// TwinCAT 3 PLC project GEMMA
// ProgramVersion: 3.1.4023.0
// libraries:
//   Tc2_Standard, * (Beckhoff Automation GmbH)
//   Tc2_System, * (Beckhoff Automation GmbH)
//   Tc3_Module, * (Beckhoff Automation GmbH)
//   VisuDialogs, * (System)
// project tree:
//   DUTs/ E_GEMMA.TcTLEO
//   / GlobalTextList.TcGTLO, ModoDescripcion.TcTLO, PlcTask.TcTTO, Visualization Manager.TcVMO (not stored)
//   POUs/Estacion/ FB_Estacion.TcPOU, FB_Coordinador_SFC.TcPOU, FB_Director.TcPOU
//   POUs/FBs/ FB_Clock.TcPOU
//   POUs/ MAIN.TcPOU
//   POUs/Tareas/ FB_CintaSituarPale_SFC.TcPOU, FB_CintaTransferirPale_SFC.TcPOU, FB_EstacionFinalizar_SFC.TcPOU, FB_EstacionPreparar_SFC.TcPOU, FB_EstacionRestaurar_SFC.TcPOU, FB_ManipuladorCargarBase_SFC.TcPOU, FB_ManipuladorDescargarBase_SFC.TcPOU, FB_PrensaPrensarRodamiento_SFC.TcPOU
//   VISUs/ TC_VISU.TcVIS

CONFIGURATION GEMMA
    RESOURCE PLC ON TwinCAT3
        TASK PlcTask(INTERVAL := T#10ms, PRIORITY := 24);
        PROGRAM MAIN WITH PlcTask : MAIN;
    END_RESOURCE
END_CONFIGURATION

// ---- DUTs/E_GEMMA.TcTLEO
{attribute 'qualified_only'}
{attribute 'strict'}
TYPE E_GEMMA :
(
    // Modos de la Guia de Estudio de los Modos de Marcha y Parada
    // [Modes du Guide d'Etude des Modes de Marche et d'Arrêt]
    // [Modes of Study Guide of the Modes of Operating and Stopping]

    // Procedimientos de parada [Les procédures d'arrets - Stop procedures]
    A1, //  0: Parada en el estado inicial [Arrêt dans etat initial - Stopped in the initial state]
    A2, //  1: Parada solicitada a final de ciclo [Arret demandé en fin de cycle - Requested end cycle stop]
    A3, //  2: Parada solicitada en un estado determinado [Arret demande dans etat determine - Requested particular state stop]
    A4, //  3: Parada obtenida [Arret obtenu - Obteined stop]
    A5, //  4: Preparacion para la recuperacion del fallo [Preparation pour remise en route apres defaillance - Preparation for the recovery of the failure]
    A6, //  5: Situando la PO en el estado inicial [Mise PO dans état initial - Set the PO in initial state]
    A7, //  6: Situando la PO en un estado determinado [Mise PO dans état déterminé - Set the PO in a certain state]

    // Procedimientos de funcionamiento [Les procédures de fonctionnement - Operating procedures]
    F1, //  7: Produccion normal [Production normale - Normal operation]
    F2, //  8: Secuencia de preparacion [Marche de preparation - Preparation sequence]
    F3, //  9: Secuencia de finalizacion [Marche de cloture - Ending sequence]
    F4, // 10: Verificacion en desorden [Marche de verification dans le desordre - Verification with no order]
    F5, // 11: Verificacion en orden [Marche de verification dans l'ordre - Verification whit order]
    F6, // 12: Secuencia de prueba [Marche de test - Test sequence]

    // Procedimientos de fallo [Les procédures en défaillances - Failure procedures]
    D1, // 13: Parada de emergencia [Arret d'urgence - Emergency stop]
    D2, // 14: Diagnostico y/o tratamiento de los fallos [Diagnostic et/ou traitement de la défaillance - Diagnosis and/or treatment of failures]
    D3  // 15: Produccion a pesar de los fallos [Production tout de même - Production despite the failures]
);
END_TYPE

// ---- POUs/MAIN.TcPOU
PROGRAM MAIN
VAR
    Estacion: FB_Estacion;
END_VAR

Estacion();

END_PROGRAM

// ---- POUs/Estacion/FB_Estacion.TcPOU
FUNCTION_BLOCK FB_Estacion
VAR_INPUT
    EstadoPausa: BOOL;
    EstadoReinicia: BOOL;
    UnidadesSolicitadas: UINT := 1;
    
    RodamientoBajo: BOOL;
    TpoCintaRetenedor: TIME := T#1S;
    TpoCintaSeparador: TIME := T#1S;
    TpoPaleEntrada: TIME := T#400ms;
    TpoPaleSalida: TIME := T#1s;
    TpoPaleTransferencia: TIME := T#1S;
    TpoPrensaHidraulico: TIME := T#2s;
    TpoPrensaProtector: TIME := T#2s;
END_VAR
VAR_OUTPUT
    CondicionInicial: BOOL := TRUE;
    UnidadesPendientes: UINT;
    UnidadesRealizadas: UINT;
    PaleCodigo: BYTE;
    
    // Entradas comunes
    PulsadorEmergencia AT %I*: BOOL;
    SelectorManual AT %I*: BOOL;
    PulsadorMarcha AT %I*: BOOL;
    PulsadorParada AT %I*: BOOL := TRUE; // Contacto normalmente cerrado
    EstacionConectada AT %I*: BOOL := TRUE;
    DetectorPresion AT %I*: BOOL := TRUE;

    PalePresencia AT %I*: BOOL;
    PaleCodigoBit0 AT %I*: BOOL;
    PaleCodigoBit1 AT %I*: BOOL;
    PaleCodigoBit2 AT %I*: BOOL;

    // Entradas espeficicas
    ManipuladorDetras AT %I*: BOOL; // Sobre el pale
    ManipuladorMedio AT %I*: BOOL := TRUE; // En la vertical
    ManipuladorDelante AT %I*: BOOL; // Sobre el punto de trasvase de la presa
    IntroductorDetras AT %I*: BOOL := TRUE;
    IntroductorDelante AT %I*: BOOL;
    ExtractorDetras AT %I*: BOOL := TRUE;
    ExtractorDelante AT %I*: BOOL;
    ProtectorAbajo AT %I*: BOOL;
    PrensadorArriba AT %I*: BOOL := TRUE;
    PrensadorAbajoAlto AT %I*: BOOL;
    PrensadorAbajoBajo AT %I*: BOOL;
    ManipuladorVacioObtenido AT %I*: BOOL;
END_VAR
VAR
    ModoAnterior: E_GEMMA;
    
    // Bloques funcionales
    CLK: FB_Clock;
    Director: FB_Director;
    Coordinador: FB_Coordinador_SFC;
    Restaurar: FB_EstacionRestaurar_SFC;
    Preparar: FB_EstacionPreparar_SFC;
    Finalizar: FB_EstacionFinalizar_SFC;
    SituarPale: FB_CintaSituarPale_SFC;
    CargarBase: FB_ManipuladorCargarBase_SFC;
    PrensarRodamiento: FB_PrensaPrensarRodamiento_SFC;
    DescargarBase: FB_ManipuladorDescargarBase_SFC;
    TransferirPale: FB_CintaTransferirPale_SFC;
    
    // Salidas comunes
    DesconectaEstacion AT %Q*: BOOL;
    LamparaAlarma AT %Q*: BOOL;
    LamparaMarcha AT %Q*: BOOL;
    AvisadorSonoro AT %Q*: BOOL;

    CintaMotorActiva AT %Q*: BOOL;
    CintaMotorInvierte AT %Q*: BOOL;
    CintaRetenedorBaja AT %Q*: BOOL;
    CintaSeparadorSube AT %Q*: BOOL;
    
    // Salidas especificas
    ManipuladorAdelante AT %Q*: BOOL; // Hacia el punto de trasvase de la prensa
    ManipuladorAtras AT %Q*: BOOL; // Hacia el pale
    IntroductorAdelante AT %Q*: BOOL;
    ExtractorAdelante AT %Q*: BOOL;
    ProtectorBaja AT %Q*: BOOL;
    PrensadorBaja AT %Q*: BOOL;
    PrensadorSube AT %Q*: BOOL;
    ManipuladorSucciona AT %Q*: BOOL;
    HidraulicoActiva AT %Q*: BOOL;
END_VAR

// MODO AUTOMATICO
CLK();

Director(
    CondicionInicial := CondicionInicial,
    CondicionMarcha := (UnidadesSolicitadas > 0) AND CondicionInicial,
    Emergencia := PulsadorEmergencia,
    Finalizada := Finalizar.Done,
    FinTarea := (UnidadesPendientes = 0),
    FinCiclo := Coordinador.Done,
    Manual := SelectorManual,
    Marcha := PulsadorMarcha,
    ParaCiclo := NOT PulsadorParada,
    Preparada := Preparar.Done,
    Reinicia := EstadoReinicia
    );

IF (Director.Modo <> E_GEMMA.F4) THEN
    // Bloques funcionales     
    Restaurar(
        SFCPause := NOT EstadoReinicia AND EstadoPausa,
        SFCReset := EstadoReinicia,
        Ack := TRUE ,
        Execute := (Director.Modo = E_GEMMA.A6) AND PulsadorMarcha,
        ManipuladorDetras := ManipuladorDetras,
        ManipuladorMedio := ManipuladorMedio,
        PrensadorArriba := PrensadorArriba
        );
        
    Preparar(
        SFCPause := NOT EstadoReinicia AND EstadoPausa,
        SFCReset := EstadoReinicia,
        Ack := (Director.Modo <> E_GEMMA.F2),
        Execute := (Director.Modo = E_GEMMA.F2),
        );

    Finalizar(
        SFCPause := NOT EstadoReinicia AND EstadoPausa,
        SFCReset := EstadoReinicia,
        Ack := (Director.Modo <> E_GEMMA.F3),
        Execute := (Director.Modo = E_GEMMA.F3),
        );
    
    Coordinador(
        UnidadesPendientes := UnidadesPendientes,
        UnidadesRealizadas := UnidadesRealizadas,
        SFCPause := NOT EstadoReinicia AND EstadoPausa,
        SFCReset := EstadoReinicia,
        Ack := TRUE,
        Execute := (Director.Modo = E_GEMMA.F1),
        PaleSituado := SituarPale.Done,
        BaseCargada := CargarBase.Done,
        RodamientoPrensado := PrensarRodamiento.Done,
        BaseDescargada := DescargarBase.Done,
        PaleTransferido := TransferirPale.Done
        );
        
    SituarPale(
        SFCPause := NOT EstadoReinicia AND EstadoPausa,
        SFCReset := EstadoReinicia,
        Ack := NOT Coordinador.SituaPale,
        Execute := Coordinador.SituaPale,
        TpoPaleEntrada := TpoPaleEntrada,
        PalePresencia := PalePresencia,
        PaleCodigoBit0 := PaleCodigoBit0,
        PaleCodigoBit1 := PaleCodigoBit1,
        PaleCodigoBit2:= PaleCodigoBit2
        );
        
    CargarBase(
        SFCPause := NOT EstadoReinicia AND EstadoPausa,
        SFCReset := EstadoReinicia,
        Ack := NOT Coordinador.CargaBase,
        Execute := Coordinador.CargaBase,
        ManipuladorDetras := ManipuladorDetras,
        ManipuladorMedio := ManipuladorMedio,
        ManipuladorDelante := ManipuladorDelante,
        ManipuladorVacioObtenido := ManipuladorVacioObtenido
        );
    
    PrensarRodamiento(
        SFCPause := NOT EstadoReinicia AND EstadoPausa,
        SFCReset := EstadoReinicia,
        Ack := NOT Coordinador.PrensaRodamiento,
        Execute := Coordinador.PrensaRodamiento,
        RodamientoBajo := RodamientoBajo,
        TpoPrensaHidraulico := TpoPrensaHidraulico,
        TpoPrensaProtector := TpoPrensaProtector,
        IntroductorDetras := IntroductorDetras,
        IntroductorDelante := IntroductorDelante,
        ExtractorDetras := ExtractorDetras,
        ExtractorDelante := ExtractorDelante,
        ProtectorAbajo := ProtectorAbajo,
        PrensadorArriba := PrensadorArriba,
        PrensadorAbajoAlto := PrensadorAbajoAlto,
        PrensadorAbajoBajo := PrensadorAbajoBajo
        );
    
    DescargarBase(
        SFCPause := NOT EstadoReinicia AND EstadoPausa,
        SFCReset := EstadoReinicia,
        Ack := NOT Coordinador.DescargaBase,
        Execute := Coordinador.DescargaBase,
        ManipuladorDetras := ManipuladorDetras,
        ManipuladorMedio := ManipuladorMedio,
        ManipuladorDelante := ManipuladorDelante,
        ManipuladorVacioObtenido := ManipuladorVacioObtenido
        );
    
    TransferirPale(
        SFCPause := NOT EstadoReinicia AND EstadoPausa,
        SFCReset := EstadoReinicia,
        Ack := NOT Coordinador.TransfierePale,
        Execute := Coordinador.TransfierePale,
        TpoCintaRetenedor := TpoCintaRetenedor,
        TpoCintaSeparador := TpoCintaSeparador,
        TpoPaleSalida := TpoPaleSalida,
        TpoPaleTransferencia := TpoPaleTransferencia,
        PalePresencia := PalePresencia
        );
    
    // Acciones
    // DesconectaEstacion :=
    LamparaAlarma := (Director.Modo = E_GEMMA.D1) OR ((Director.Modo = E_GEMMA.A6) AND CLK.Q);
    LamparaMarcha := Director.Produccion OR ((Director.Modo = E_GEMMA.A1) AND CLK.Q);
    AvisadorSonoro := ((Director.Modo = E_GEMMA.F2) AND CLK.Q) OR (Director.Modo = E_GEMMA.F3); 

    CintaMotorActiva := NOT EstadoPausa AND (SituarPale.CintaMotorActiva OR TransferirPale.CintaMotorActiva);
    // CintaMotorInvierte :=
    CintaRetenedorBaja:= TransferirPale.CintaRetenedorBaja;
    CintaSeparadorSube :=TransferirPale.CintaSeparadorSube;
    ManipuladorAdelante := CargarBase.ManipuladorAdelante OR DescargarBase.ManipuladorAdelante OR Restaurar.ManipuladorAdelante;
    ManipuladorAtras := CargarBase.ManipuladorAtras OR DescargarBase.ManipuladorAtras OR Restaurar.ManipuladorAtras;
    IntroductorAdelante := PrensarRodamiento.IntroductorAdelante;
    ExtractorAdelante := PrensarRodamiento.ExtractorAdelante;
    ProtectorBaja := PrensarRodamiento.ProtectorBaja;
    PrensadorBaja := PrensarRodamiento.PrensadorBaja;
    PrensadorSube := PrensarRodamiento.PrensadorSube OR Restaurar.PrensadorSube;
    ManipuladorSucciona := CargarBase.ManipuladorSucciona OR DescargarBase.ManipuladorSucciona;
    HidraulicoActiva := PrensarRodamiento.HidraulicoActiva;
END_IF

// Parametros de Salida
CondicionInicial := EstacionConectada AND ManipuladorMedio AND IntroductorDetras AND ExtractorDetras AND PrensadorArriba;

// Al iniciar una tarea (abandonar modo A1) se actualiza las unidades pendientes
IF ((ModoAnterior = E_GEMMA.A1) AND (Director.Modo <> E_GEMMA.A1) AND (UnidadesPendientes = 0)) THEN
    UnidadesPendientes := UnidadesSolicitadas;
END_IF
 
IF (Director.Modo <> E_GEMMA.F4) THEN
    PaleCodigo := SituarPale.PaleCodigo;
ELSE 
    PaleCodigo.0 := PaleCodigoBit0;
    PaleCodigo.1 := PaleCodigoBit1;
    PaleCodigo.2 := PaleCodigoBit2;
END_IF

// ACTULIZACION DE IMAGENES
ModoAnterior := Director.Modo;

END_FUNCTION_BLOCK

// ---- POUs/FBs/FB_Clock.TcPOU
FUNCTION_BLOCK FB_Clock
(*
Square wave oscillator

Copyright (c) 2009-2017 victortorreslopez

GNU General Public License

Version history
2.1, 2017/03/15, VTL: style review (PLCopen Coding Guidelines)
2.0, 2014/12/29, VTL: complete review
1.0, 2009/11/06, VTL: first release
0.0, 2009/11/06, VTL: alfa release
*)
VAR_INPUT
  EN: BOOL := TRUE;	(* ENabled *)
  PT: TIME := T#500ms; (* Semicycle time *)
END_VAR
VAR_OUTPUT
  ET: TIME; (* Elapsed time *)
  Q: BOOL; (* Square wave *)
END_VAR
VAR
  Timer: TON; (* Auto-pilot timer *)
END_VAR

(* OUTPUT FUNCTION *)
IF Timer.Q THEN
  Q := NOT Q;
END_IF

(* FUNCTION BLOCKS *)
Timer(IN := EN AND NOT Timer.Q, PT := PT, ET => ET);

END_FUNCTION_BLOCK

// ---- POUs/Estacion/FB_Director.TcPOU
FUNCTION_BLOCK FB_Director
VAR_INPUT
    CondicionInicial: BOOL; // Condiciones materiales necesarias para iniciar la produccion
    CondicionMarcha: BOOL; // Condiciones logicas necesarias para iniciar la produccion
    Emergencia: BOOL;
    Finalizada: BOOL;
    FinTarea: BOOL;
    FinCiclo: BOOL;
    Manual: BOOL;
    Marcha: BOOL;
    ParaCiclo: BOOL;
    Preparada: BOOL;
    Reinicia: BOOL;
END_VAR
VAR_OUTPUT
    Modo: E_GEMMA := E_GEMMA.A6;

    Defecto: BOOL; // Procedimientos de defecto
    Funcionamiento: BOOL; // Procedimientos de funcionamiento
    Parada: BOOL; // Procedimientos de parada
    Produccion: BOOL; // Procedimientos que proporcionan valor añadido
END_VAR

// FUNCION DE ESTADO
IF Emergencia THEN
    Modo := E_GEMMA.D1;
ELSIF Reinicia THEN
    Modo := E_GEMMA.A6;
ELSE
    CASE Modo OF
        // Procedimientos de parada
        E_GEMMA.A1: // Parada en el estado inicial
            IF NOT CondicionInicial THEN
                Modo := E_GEMMA.A6;
            ELSIF Manual THEN
                Modo := E_GEMMA.F4;
            ELSIF (CondicionMarcha AND Marcha) THEN
                Modo := E_GEMMA.F2;
            END_IF
        E_GEMMA.A2: // Parada solicitada a final de ciclo
            IF FinCiclo THEN
                Modo := E_GEMMA.A1;
            END_IF
        E_GEMMA.A3: // Parada solicitada en un estado determinado 
            ;
        E_GEMMA.A4: // Parada obtenida 
            ;
        E_GEMMA.A5: // Preparando de reanudacion tras el fallo 
            ;
        E_GEMMA.A6: // Situando la PO en el estado inicial 
            IF CondicionInicial THEN
                Modo := E_GEMMA.A1;
            ELSIF Manual THEN
                Modo := E_GEMMA.F4;
            END_IF
        E_GEMMA.A7: // Situando la PO en un estado determinado 
            ;

        // Procedimientos de funcionamiento 
        E_GEMMA.F1: // Produccion normal 
            IF FinTarea THEN
                Modo := E_GEMMA.F3;
            ELSIF ParaCiclo THEN
                Modo := E_GEMMA.A2;
            END_IF
        E_GEMMA.F2: // Secuencia de preparacion 
            IF Preparada THEN
                Modo := E_GEMMA.F1;
            END_IF
        E_GEMMA.F3: // Secuencia de finalizacion 
            IF Finalizada THEN
                Modo := E_GEMMA.A1;
            END_IF
        E_GEMMA.F4: // Verificacion sin orden 
            IF NOT Manual THEN
                Modo := E_GEMMA.A6;
            END_IF
        E_GEMMA.F5: // Verificacion en orden 
            ;
        E_GEMMA.F6: // Prueba 
            ;

        // Procedimientos de defecto 
        E_GEMMA.D1: // Parada de emergencia 
            IF NOT Emergencia THEN
                Modo := E_GEMMA.A6;
            END_IF
        E_GEMMA.D2: // Diagnostico/tratamiento de los fallos 
            ;
        E_GEMMA.D3: // Produccion a pesar de los fallos 
            ;
    END_CASE
END_IF

// PARAMETROS DE SALIDA 
Defecto := (Modo >= E_GEMMA.D1) AND (Modo <= E_GEMMA.D3);
Funcionamiento:= (Modo >= E_GEMMA.F1) AND (Modo <= E_GEMMA.F6);
Parada := (Modo >= E_GEMMA.A1) AND (Modo <= E_GEMMA.A7);
Produccion := (Modo = E_GEMMA.A2) OR (Modo = E_GEMMA.A3) OR (Modo = E_GEMMA.F1) 
    OR (Modo = E_GEMMA.F2) OR (Modo = E_GEMMA.F3) OR (Modo = E_GEMMA.F5)
    OR (Modo = E_GEMMA.F6) OR (Modo = E_GEMMA.D3);

END_FUNCTION_BLOCK

// ---- POUs/Estacion/FB_Coordinador_SFC.TcPOU
FUNCTION_BLOCK FB_Coordinador_SFC
VAR_IN_OUT
    UnidadesPendientes: UINT;
    UnidadesRealizadas: UINT;
END_VAR
VAR_INPUT
    // SFC-Flags
    SFCPause: BOOL;
    SFCReset: BOOL;
    
    // Indicadores de sincronizacion
    Ack: BOOL := TRUE;
    Execute: BOOL;
    
    // Parametros de sincronizacion
    PaleSituado: BOOL;
    BaseCargada: BOOL;
    RodamientoPrensado: BOOL;
    BaseDescargada: BOOL;
    PaleTransferido: BOOL;
END_VAR
VAR_OUTPUT
    // Indicadores de sincronizacion
    Done: BOOL;
    Ready: BOOL;

    // Parametros de sincronizacion
    SituaPale: BOOL;
    CargaBase: BOOL;
    PrensaRodamiento: BOOL;
    DescargaBase: BOOL;
    TransfierePale: BOOL;
END_VAR
VAR
END_VAR

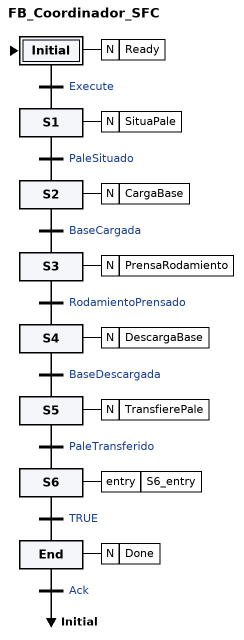
INITIAL_STEP Initial:
    Ready(N);
END_STEP
TRANSITION FROM Initial TO S1
    := Execute;
END_TRANSITION
STEP S1:
    SituaPale(N);
END_STEP
TRANSITION FROM S1 TO S2
    := PaleSituado;
END_TRANSITION
STEP S2:
    CargaBase(N);
END_STEP
TRANSITION FROM S2 TO S3
    := BaseCargada;
END_TRANSITION
STEP S3:
    PrensaRodamiento(N);
END_STEP
TRANSITION FROM S3 TO S4
    := RodamientoPrensado;
END_TRANSITION
STEP S4:
    DescargaBase(N);
END_STEP
TRANSITION FROM S4 TO S5
    := BaseDescargada;
END_TRANSITION
STEP S5:
    TransfierePale(N);
END_STEP
TRANSITION FROM S5 TO S6
    := PaleTransferido;
END_TRANSITION
STEP S6:
    S6_entry(P1);  // entry action
END_STEP
TRANSITION FROM S6 TO End
    := TRUE;
END_TRANSITION
STEP End:
    Done(N);
END_STEP
TRANSITION FROM End TO Initial
    := Ack;
END_TRANSITION

ACTION S6_entry:
// Al completar la transferencia del pale
UnidadesRealizadas := UnidadesRealizadas + 1;

IF (UnidadesPendientes > 0) THEN
    UnidadesPendientes := UnidadesPendientes - 1;
END_IF
END_ACTION

END_FUNCTION_BLOCK

// ---- POUs/Tareas/FB_EstacionRestaurar_SFC.TcPOU
FUNCTION_BLOCK FB_EstacionRestaurar_SFC
VAR_INPUT
    // SFC-Flags
    SFCPause: BOOL;
    SFCReset: BOOL;
    
    // Indicadores de sincronizacion
    Ack: BOOL := TRUE;
    Execute: BOOL;
    
    // Entradas
    ManipuladorDetras: BOOL; // Sobre el pale
    ManipuladorMedio: BOOL := TRUE; // En la vertical
    PrensadorArriba: BOOL := TRUE;
END_VAR
VAR_OUTPUT
    // Indicadores de sincronizacion
    Done: BOOL;
    Ready: BOOL;
    
    // Salidas
    ManipuladorAdelante: BOOL; // Hacia el punto de trasvase de la prensa
    ManipuladorAtras: BOOL; // Hacia el pale
    PrensadorSube: BOOL;    
END_VAR
VAR
END_VAR

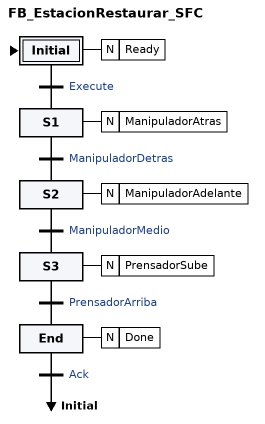
INITIAL_STEP Initial:
    Ready(N);
END_STEP
TRANSITION FROM Initial TO S1
    := Execute;
END_TRANSITION
STEP S1:
    ManipuladorAtras(N);
END_STEP
TRANSITION FROM S1 TO S2
    := ManipuladorDetras;
END_TRANSITION
STEP S2:
    ManipuladorAdelante(N);
END_STEP
TRANSITION FROM S2 TO S3
    := ManipuladorMedio;
END_TRANSITION
STEP S3:
    PrensadorSube(N);
END_STEP
TRANSITION FROM S3 TO End
    := PrensadorArriba;
END_TRANSITION
STEP End:
    Done(N);
END_STEP
TRANSITION FROM End TO Initial
    := Ack;
END_TRANSITION

END_FUNCTION_BLOCK

// ---- POUs/Tareas/FB_EstacionPreparar_SFC.TcPOU
FUNCTION_BLOCK FB_EstacionPreparar_SFC
VAR_INPUT
    // SFC-Flags
    SFCPause: BOOL;
    SFCReset: BOOL;
    
    // Indicadores de sincronizacion
    Ack: BOOL := TRUE;
    Execute: BOOL;
    
    // Parametros
    TpoPreparacion: TIME := T#3S;
END_VAR
VAR_OUTPUT
    // Indicadores de sincronizacion
    Done: BOOL;
    Ready: BOOL;
END_VAR
VAR
END_VAR

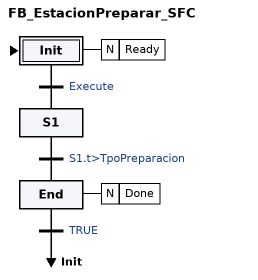
INITIAL_STEP Init:
    Ready(N);
END_STEP
TRANSITION FROM Init TO S1
    := Execute;
END_TRANSITION
STEP S1:
END_STEP
TRANSITION FROM S1 TO End
    := S1.t>TpoPreparacion;
END_TRANSITION
STEP End:
    Done(N);
END_STEP
TRANSITION FROM End TO Init
    := TRUE;
END_TRANSITION

END_FUNCTION_BLOCK

// ---- POUs/Tareas/FB_EstacionFinalizar_SFC.TcPOU
FUNCTION_BLOCK FB_EstacionFinalizar_SFC
VAR_INPUT
    // SFC-Flags
    SFCPause: BOOL;
    SFCReset: BOOL;
    
    // Indicadores de sincronizacion
    Ack: BOOL := TRUE;
    Execute: BOOL;
    
    // Parametros
    TpoFinalizacion: TIME := T#1S;
END_VAR
VAR_OUTPUT
    // Indicadores de sincronizacion
    Done: BOOL;
    Ready: BOOL;
END_VAR
VAR
END_VAR

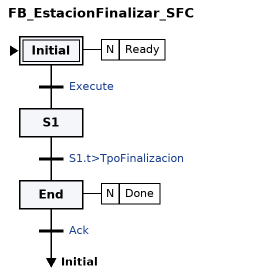
INITIAL_STEP Initial:
    Ready(N);
END_STEP
TRANSITION FROM Initial TO S1
    := Execute;
END_TRANSITION
STEP S1:
END_STEP
TRANSITION FROM S1 TO End
    := S1.t>TpoFinalizacion;
END_TRANSITION
STEP End:
    Done(N);
END_STEP
TRANSITION FROM End TO Initial
    := Ack;
END_TRANSITION

END_FUNCTION_BLOCK

// ---- POUs/Tareas/FB_CintaSituarPale_SFC.TcPOU
FUNCTION_BLOCK FB_CintaSituarPale_SFC
VAR_INPUT
    // SFC-Flags
    SFCPause: BOOL;
    SFCReset: BOOL;
    
    // Indicadores de sincronizacion
    Ack: BOOL := TRUE;
    Execute: BOOL;
    
    // Parametros
    TpoPaleEntrada: TIME := T#400MS;
    
    // Entradas
    PalePresencia: BOOL;
    PaleCodigoBit0: BOOL;
    PaleCodigoBit1: BOOL;
    PaleCodigoBit2: BOOL;    
END_VAR
VAR_OUTPUT
    // Indicadores de sincronizacion
    Done: BOOL;
    Ready: BOOL;
    
    // Parametros
    PaleCodigo: BYTE;
    
    // Salidas
    CintaMotorActiva: BOOL;
END_VAR
VAR
END_VAR

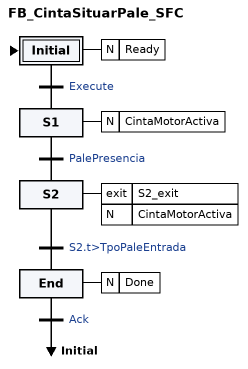
INITIAL_STEP Initial:
    Ready(N);
END_STEP
TRANSITION FROM Initial TO S1
    := Execute;
END_TRANSITION
STEP S1:
    CintaMotorActiva(N);
END_STEP
TRANSITION FROM S1 TO S2
    := PalePresencia;
END_TRANSITION
STEP S2:
    S2_exit(P0);  // exit action
    CintaMotorActiva(N);
END_STEP
TRANSITION FROM S2 TO End
    := S2.t>TpoPaleEntrada;
END_TRANSITION
STEP End:
    Done(N);
END_STEP
TRANSITION FROM End TO Initial
    := Ack;
END_TRANSITION

ACTION S2_exit:
PaleCodigo.0 := PaleCodigoBit0;
PaleCodigo.1 := PaleCodigoBit1;
PaleCodigo.2 := PaleCodigoBit2;
END_ACTION

END_FUNCTION_BLOCK

// ---- POUs/Tareas/FB_ManipuladorCargarBase_SFC.TcPOU
FUNCTION_BLOCK FB_ManipuladorCargarBase_SFC
VAR_INPUT
    // SFC-Flags
    SFCPause: BOOL;
    SFCReset: BOOL;
    
    // Indicadores de sincronizacion
    Ack: BOOL := TRUE;
    Execute: BOOL;
    
    // Entradas
    ManipuladorDetras: BOOL; // Sobre el pale
    ManipuladorMedio: BOOL := TRUE; // En la vertical
    ManipuladorDelante: BOOL; // Sobre el punto de trasvase de la presa\
    ManipuladorVacioObtenido: BOOL;
END_VAR
VAR_OUTPUT
    // Indicadores de sincronizacion
    Done: BOOL;
    Ready: BOOL;

    // Salidas
    ManipuladorAdelante: BOOL; // Hacia el punto de trasvase de la prensa
    ManipuladorAtras: BOOL; // Hacia el pale
    ManipuladorSucciona: BOOL;
END_VAR
VAR
END_VAR

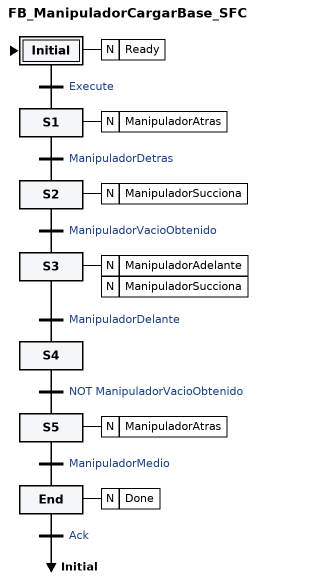
INITIAL_STEP Initial:
    Ready(N);
END_STEP
TRANSITION FROM Initial TO S1
    := Execute;
END_TRANSITION
STEP S1:
    ManipuladorAtras(N);
END_STEP
TRANSITION FROM S1 TO S2
    := ManipuladorDetras;
END_TRANSITION
STEP S2:
    ManipuladorSucciona(N);
END_STEP
TRANSITION FROM S2 TO S3
    := ManipuladorVacioObtenido;
END_TRANSITION
STEP S3:
    ManipuladorAdelante(N);
    ManipuladorSucciona(N);
END_STEP
TRANSITION FROM S3 TO S4
    := ManipuladorDelante;
END_TRANSITION
STEP S4:
END_STEP
TRANSITION FROM S4 TO S5
    := NOT ManipuladorVacioObtenido;
END_TRANSITION
STEP S5:
    ManipuladorAtras(N);
END_STEP
TRANSITION FROM S5 TO End
    := ManipuladorMedio;
END_TRANSITION
STEP End:
    Done(N);
END_STEP
TRANSITION FROM End TO Initial
    := Ack;
END_TRANSITION

END_FUNCTION_BLOCK

// ---- POUs/Tareas/FB_PrensaPrensarRodamiento_SFC.TcPOU
FUNCTION_BLOCK FB_PrensaPrensarRodamiento_SFC
VAR_INPUT
    // SFC-Flags
    SFCPause: BOOL;
    SFCReset: BOOL;
    
    // Indicadores de sincronizacion
    Ack: BOOL := TRUE;
    Execute: BOOL;
    
    // Parametros
    RodamientoBajo: BOOL;
    TpoPrensaHidraulico: TIME := T#2S;
    TpoPrensaProtector: TIME := T#2S;
    
    // Entradas
    IntroductorDetras: BOOL := TRUE;
    IntroductorDelante: BOOL;
    ExtractorDetras: BOOL := TRUE;
    ExtractorDelante: BOOL;
    ProtectorAbajo: BOOL;
    PrensadorArriba: BOOL := TRUE;
    PrensadorAbajoAlto: BOOL;
    PrensadorAbajoBajo: BOOL;
END_VAR
VAR_OUTPUT
    // Indicadores de sincronizacion
    Done: BOOL;
    Ready: BOOL;
    
    // Salidas
    IntroductorAdelante: BOOL;
    ExtractorAdelante: BOOL;
    ProtectorBaja: BOOL;
    PrensadorBaja: BOOL;
    PrensadorSube: BOOL;
    HidraulicoActiva: BOOL;
END_VAR
VAR
END_VAR

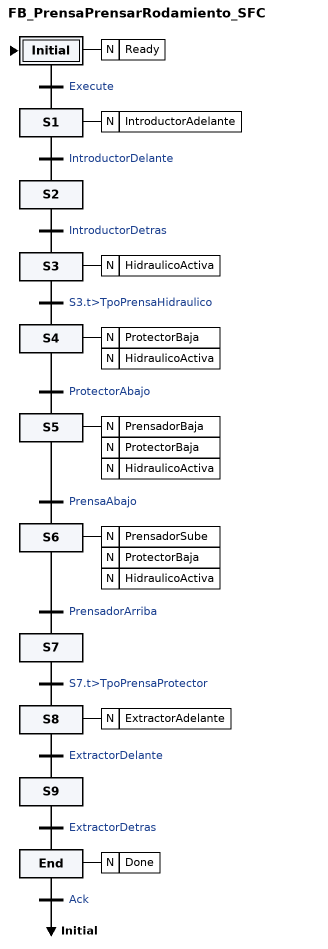
INITIAL_STEP Initial:
    Ready(N);
END_STEP
TRANSITION FROM Initial TO S1
    := Execute;
END_TRANSITION
STEP S1:
    IntroductorAdelante(N);
END_STEP
TRANSITION FROM S1 TO S2
    := IntroductorDelante;
END_TRANSITION
STEP S2:
END_STEP
TRANSITION FROM S2 TO S3
    := IntroductorDetras;
END_TRANSITION
STEP S3:
    HidraulicoActiva(N);
END_STEP
TRANSITION FROM S3 TO S4
    := S3.t>TpoPrensaHidraulico;
END_TRANSITION
STEP S4:
    ProtectorBaja(N);
    HidraulicoActiva(N);
END_STEP
TRANSITION FROM S4 TO S5
    := ProtectorAbajo;
END_TRANSITION
STEP S5:
    PrensadorBaja(N);
    ProtectorBaja(N);
    HidraulicoActiva(N);
END_STEP
TRANSITION FROM S5 TO S6
    := PrensaAbajo;
END_TRANSITION
STEP S6:
    PrensadorSube(N);
    ProtectorBaja(N);
    HidraulicoActiva(N);
END_STEP
TRANSITION FROM S6 TO S7
    := PrensadorArriba;
END_TRANSITION
STEP S7:
END_STEP
TRANSITION FROM S7 TO S8
    := S7.t>TpoPrensaProtector;
END_TRANSITION
STEP S8:
    ExtractorAdelante(N);
END_STEP
TRANSITION FROM S8 TO S9
    := ExtractorDelante;
END_TRANSITION
STEP S9:
END_STEP
TRANSITION FROM S9 TO End
    := ExtractorDetras;
END_TRANSITION
STEP End:
    Done(N);
END_STEP
TRANSITION FROM End TO Initial
    := Ack;
END_TRANSITION

TRANSITION PrensaAbajo:
// La prensa baja mas o menos dependiendo del tipo de rodamiento
(NOT RodamientoBajo AND PrensadorAbajoAlto) OR (RodamientoBajo AND PrensadorAbajoBajo)
END_TRANSITION

END_FUNCTION_BLOCK

// ---- POUs/Tareas/FB_ManipuladorDescargarBase_SFC.TcPOU
FUNCTION_BLOCK FB_ManipuladorDescargarBase_SFC
VAR_INPUT
    // SFC-Flags
    SFCPause: BOOL;
    SFCReset: BOOL;
    
    // Indicadores de sincronizacion
    Ack: BOOL := TRUE;
    Execute: BOOL;
    
    // Entradas
    ManipuladorDetras: BOOL; // Sobre el pale
    ManipuladorMedio: BOOL := TRUE; // En la vertical
    ManipuladorDelante: BOOL; // Sobre el punto de trasvase de la presa
    ManipuladorVacioObtenido: BOOL;
END_VAR
VAR_OUTPUT
    // Indicadores de sincronizacion
    Done: BOOL;
    Ready: BOOL;
    
    // Salidas
    ManipuladorAdelante: BOOL; // Hacia el punto de trasvase de la prensa
    ManipuladorAtras: BOOL; // Hacia el pale
    ManipuladorSucciona: BOOL;
END_VAR
VAR
END_VAR

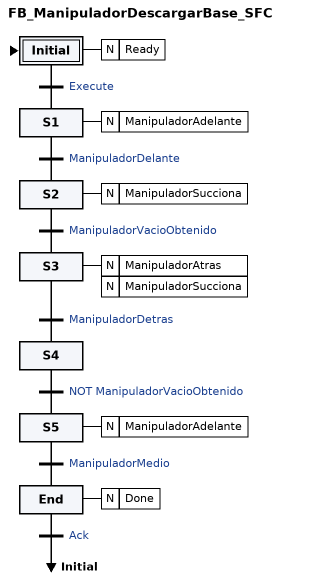
INITIAL_STEP Initial:
    Ready(N);
END_STEP
TRANSITION FROM Initial TO S1
    := Execute;
END_TRANSITION
STEP S1:
    ManipuladorAdelante(N);
END_STEP
TRANSITION FROM S1 TO S2
    := ManipuladorDelante;
END_TRANSITION
STEP S2:
    ManipuladorSucciona(N);
END_STEP
TRANSITION FROM S2 TO S3
    := ManipuladorVacioObtenido;
END_TRANSITION
STEP S3:
    ManipuladorAtras(N);
    ManipuladorSucciona(N);
END_STEP
TRANSITION FROM S3 TO S4
    := ManipuladorDetras;
END_TRANSITION
STEP S4:
END_STEP
TRANSITION FROM S4 TO S5
    := NOT ManipuladorVacioObtenido;
END_TRANSITION
STEP S5:
    ManipuladorAdelante(N);
END_STEP
TRANSITION FROM S5 TO End
    := ManipuladorMedio;
END_TRANSITION
STEP End:
    Done(N);
END_STEP
TRANSITION FROM End TO Initial
    := Ack;
END_TRANSITION

END_FUNCTION_BLOCK

// ---- POUs/Tareas/FB_CintaTransferirPale_SFC.TcPOU
FUNCTION_BLOCK FB_CintaTransferirPale_SFC
VAR_INPUT
    // SFC-Flags
    SFCPause: BOOL;
    SFCReset: BOOL;
    
    // Indicadores de sincronizacion
    Ack: BOOL := TRUE;
    Execute: BOOL;
    
    // Parametros
    TpoCintaRetenedor: TIME := T#1S;
    TpoCintaSeparador: TIME := T#1S;
    TpoPaleSalida: TIME := T#1S;
    TpoPaleTransferencia: TIME := T#1S;
    
    // Entradas
    PalePresencia: BOOL;
END_VAR
VAR_OUTPUT
    // Indicadores de sincronizacion
    Done: BOOL;
    Ready: BOOL;
    // Salidas
    CintaMotorActiva: BOOL;
    CintaRetenedorBaja: BOOL;
    CintaSeparadorSube: BOOL;
END_VAR
VAR
END_VAR

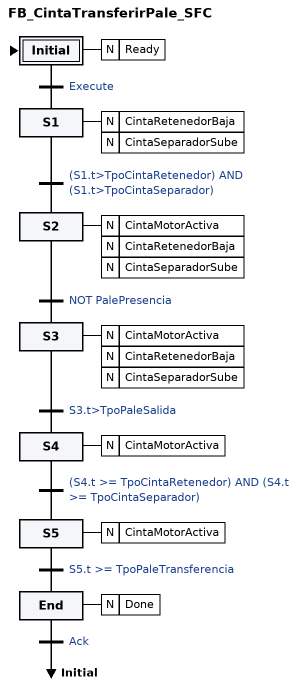
INITIAL_STEP Initial:
    Ready(N);
END_STEP
TRANSITION FROM Initial TO S1
    := Execute;
END_TRANSITION
STEP S1:
    CintaRetenedorBaja(N);
    CintaSeparadorSube(N);
END_STEP
TRANSITION FROM S1 TO S2
    := (S1.t>TpoCintaRetenedor) AND (S1.t>TpoCintaSeparador);
END_TRANSITION
STEP S2:
    CintaMotorActiva(N);
    CintaRetenedorBaja(N);
    CintaSeparadorSube(N);
END_STEP
TRANSITION FROM S2 TO S3
    := NOT PalePresencia;
END_TRANSITION
STEP S3:
    CintaMotorActiva(N);
    CintaRetenedorBaja(N);
    CintaSeparadorSube(N);
END_STEP
TRANSITION FROM S3 TO S4
    := S3.t>TpoPaleSalida;
END_TRANSITION
STEP S4:
    CintaMotorActiva(N);
END_STEP
TRANSITION FROM S4 TO S5
    := (S4.t >= TpoCintaRetenedor) AND (S4.t >= TpoCintaSeparador);
END_TRANSITION
STEP S5:
    CintaMotorActiva(N);
END_STEP
TRANSITION FROM S5 TO End
    := S5.t >= TpoPaleTransferencia;
END_TRANSITION
STEP End:
    Done(N);
END_STEP
TRANSITION FROM End TO Initial
    := Ack;
END_TRANSITION

END_FUNCTION_BLOCK

// ---- GlobalTextList.TcGTLO
TEXTLIST GlobalTextList
  939 = '%d'
  602 = '%s'
  833 = '+'
  832 = '-'
  402 = '.0'
  16 = '.1'
  415 = '.2'
  831 = '0'
  830 = '1'
  834 = '2'
  3 = '2023'
  827 = '3'
  39 = '4'
  583 = 'A'
  743 = 'Alto'
  739 = 'B'
  984 = 'Bajo'
  782 = 'C'
  941 = 'Cargador Cilindro'
  486 = 'Cargador Eyector'
  228 = 'CI'
  912 = 'Cinta Motor'
  423 = 'Cinta Retenedor'
  852 = 'Cinta Separador'
  951 = 'Conectada'
  122 = 'cp'
  419 = 'Código Palé'
  820 = 'D'
  1323 = 'Desconecta'
  469 = 'E'
  695 = 'Emergencia'
  87 = 'Entrada Palé'
  585 = 'Estructurado'
  902 = 'Extractor'
  896 = 'FMS-203'
  243 = 'GEMMA'
  489 = 'Grupo Hidráulico'
  222 = 'H'
  129 = 'Hidráulico'
  524 = 'Introductor'
  372 = 'ISA'
  531 = 'KM'
  927 = 'L. Alarma'
  664 = 'L. Marcha'
  537 = 'Manipulador'
  287 = 'Manipulador Cilindro'
  139 = 'Manipulador Eyector'
  923 = 'Manual'
  332 = 'Modo'
  544 = 'P. Marcha'
  15 = 'P. Parada'
  438 = 'PANEL'
  584 = 'PARÁMETROS'
  37 = 'Pausa'
  513 = 'Pendientes'
  284 = 'PLANTA'
  676 = 'pp'
  424 = 'PRENSADO HIDRÁULICO DEL RODAMIENTO'
  64 = 'Prensador'
  366 = 'Presostato'
  258 = 'Protector'
  171 = 'R'
  915 = 'Realizadas'
  328 = 'Reposo'
  621 = 'Reset'
  190 = 'Retenedor'
  248 = 'S'
  949 = 'Salida Palé'
  693 = 'Separador'
  333 = 'Solicitadas'
  390 = 'TAREA'
  569 = 'Transf. Palé'
  441 = 'V'
END_TEXTLIST

// ---- ModoDescripcion.TcTLO
TEXTLIST ModoDescripcion
  0 = 'Parada en el estado inicial'
  1 = 'Parada a final de ciclo'
  2 = 'Parada pedida'
  3 = 'Parada obtenida'
  4 = 'Recuperación del defecto'
  5 = 'Puesta en el estado inicial'
  6 = 'Puesta en un estado determinado'
  7 = 'Produccion normal'
  8 = 'Marchas de preparación'
  9 = 'Marchas de cierre'
  10 = 'M. verificacion en desorden'
  11 = 'M. verificacion en orden'
  12 = 'Marchas de prueba'
  13 = 'Emergencia'
  14 = 'Tratamiento de los defectos'
  15 = 'Producción con defectos'
   = ''
END_TEXTLIST

// ---- VISUs/TC_VISU.TcVIS
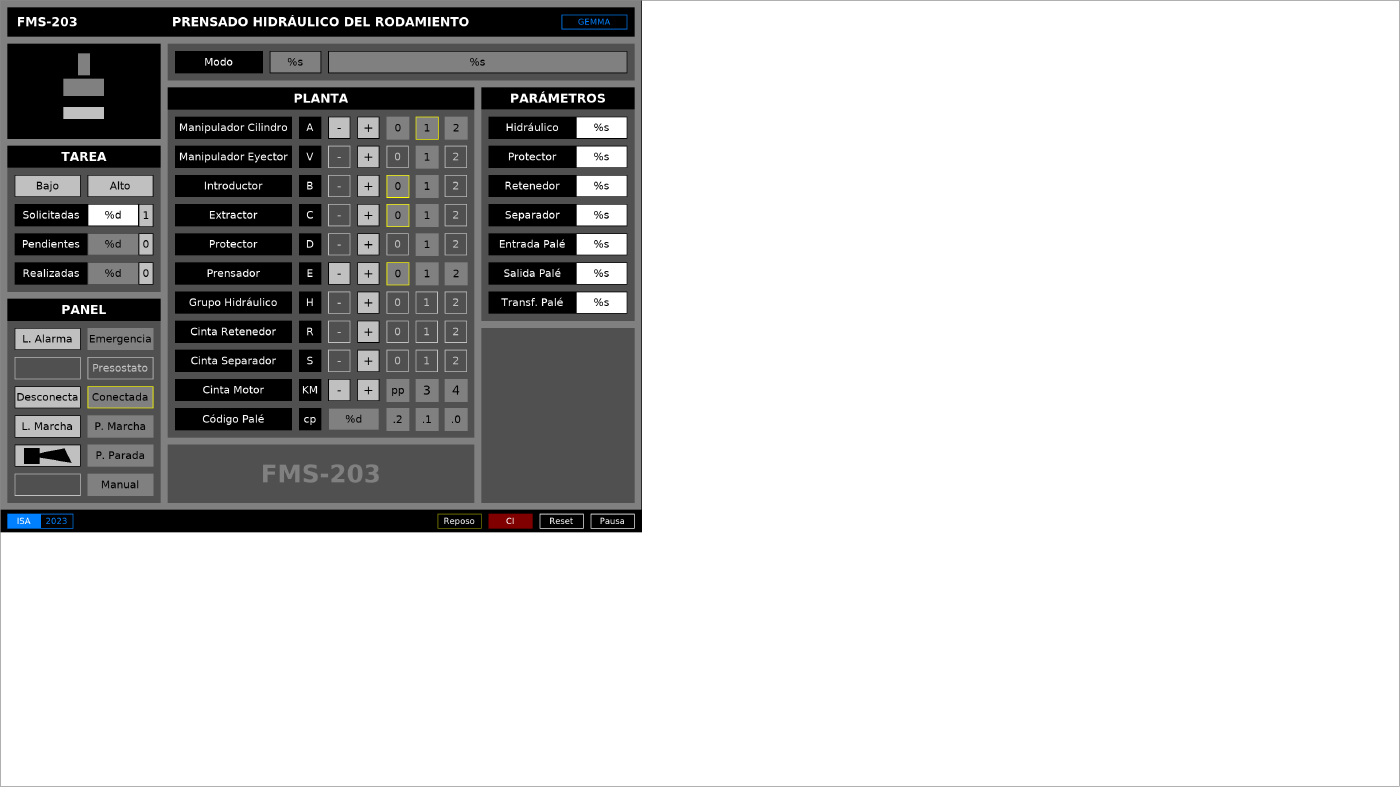
VISUALIZATION TC_VISU  // 1920x1080
    Rectangle (120,610 90x30)
    Rectangle (0,0 880x700)
    Rectangle (230,150 420x450)
    Rectangle (10,440 210x250)
    Rectangle (10,10 860x40), "PRENSADO HIDRÁULICO DEL RODAMIENTO"
    Rectangle (770,20 90x20), "GEMMA"
    Rectangle (10,60 210x130)
    Rectangle (230,120 420x30), "PLANTA"
    Rectangle (240,160 160x30), "Manipulador Cilindro"
    Rectangle (410,160 30x30), "A"
    Rectangle (450,160 30x30), "-"
    Rectangle (490,160 30x30), "+"
    Rectangle (530,160 30x30), "0"
    Rectangle (570,160 30x30), "1"
    Rectangle (610,160 30x30), "2"
    Rectangle (530,160 31x31), "0", colour toggle: MAIN.Estacion.ManipuladorDetras
        toggle MAIN.Estacion.ManipuladorDetras
    Rectangle (490,160 30x30), "+", colour toggle: MAIN.Estacion.ManipuladorAdelante
        toggle MAIN.Estacion.ManipuladorAdelante
    Rectangle (570,160 31x31), "1", colour toggle: MAIN.Estacion.ManipuladorMedio
        toggle MAIN.Estacion.ManipuladorMedio
    Rectangle (240,240 160x30), "Introductor"
    Rectangle (410,240 30x30), "B"
    Rectangle (10,410 210x30), "PANEL"
    Rectangle (20,450 90x30)
    Rectangle (0,700 880x30)
    Rectangle (55,705 45x20), "2023"
    Rectangle (10,705 45x20), "ISA"
    Rectangle (20,490 90x30)
    Rectangle (120,490 90x30), "Presostato"
    Rectangle (20,530 90x30)
    Rectangle (20,570 90x30)
    Rectangle (20,610 90x30)
    Rectangle (20,650 90x30)
    Rectangle (20,450 90x30), "L. Alarma", colour toggle: MAIN.Estacion.LamparaAlarma
        tap MAIN.Estacion.LamparaAlarma
    Rectangle (20,530 90x30), "Desconecta", colour toggle: MAIN.Estacion.DesconectaEstacion
        tap MAIN.Estacion.DesconectaEstacion
    Rectangle (20,570 90x30), "L. Marcha", colour toggle: MAIN.Estacion.LamparaMarcha
        tap MAIN.Estacion.LamparaMarcha
    Rectangle (20,610 90x30), colour toggle: MAIN.Estacion.AvisadorSonoro
        tap MAIN.Estacion.AvisadorSonoro
    Rectangle (120,450 90x30), colour toggle: MAIN.Estacion.PulsadorEmergencia
        toggle MAIN.Estacion.PulsadorEmergencia
    Rectangle (120,570 90x30)
    Rectangle (120,530 90x30)
    Rectangle (120,650 90x30)
    Rectangle (240,280 160x30), "Extractor"
    Rectangle (410,280 30x30), "C"
    Rectangle (240,320 160x30), "Protector"
    Rectangle (410,320 30x30), "D"
    Rectangle (240,360 160x30), "Prensador"
    Rectangle (410,360 30x30), "E"
    Rectangle (240,200 160x30), "Manipulador Eyector"
    Rectangle (410,200 30x30), "V"
    Rectangle (240,400 160x30), "Grupo Hidráulico"
    Rectangle (410,400 30x30), "H"
    Rectangle (240,440 160x30), "Cinta Retenedor"
    Rectangle (410,440 30x30), "R"
    Rectangle (240,480 160x30), "Cinta Separador"
    Rectangle (410,480 30x30), "S"
    Rectangle (240,520 160x30), "Cinta Motor"
    Rectangle (410,520 30x30), "KM"
    Rectangle (240,560 160x30), "Código Palé"
    Rectangle (410,560 30x30), "cp"
    Rectangle (230,610 420x80), "FMS-203"
    Rectangle (450,240 30x30), "-"
    Rectangle (490,240 30x30), "+"
    Rectangle (530,240 30x30), "0"
    Rectangle (570,240 30x30), "1"
    Rectangle (610,240 30x30), "2"
    Rectangle (530,240 31x31), "0", colour toggle: MAIN.Estacion.IntroductorDetras
        toggle MAIN.Estacion.IntroductorDetras
    Rectangle (490,240 30x30), "+", colour toggle: MAIN.Estacion.IntroductorAdelante
        toggle MAIN.Estacion.IntroductorAdelante
    Rectangle (570,240 31x31), "1", colour toggle: MAIN.Estacion.IntroductorDelante
        toggle MAIN.Estacion.IntroductorDelante
    Rectangle (450,280 30x30), "-"
    Rectangle (490,280 30x30), "+"
    Rectangle (530,280 30x30), "0"
    Rectangle (570,280 30x30), "1"
    Rectangle (610,280 30x30), "2"
    Rectangle (530,280 31x31), "0", colour toggle: MAIN.Estacion.ExtractorDetras
        toggle MAIN.Estacion.ExtractorDetras
    Rectangle (490,280 30x30), "+", colour toggle: MAIN.Estacion.ExtractorAdelante
        toggle MAIN.Estacion.ExtractorAdelante
    Rectangle (570,280 31x31), "1", colour toggle: MAIN.Estacion.ExtractorDelante
        toggle MAIN.Estacion.ExtractorDelante
    Rectangle (450,320 30x30), "-"
    Rectangle (490,320 30x30), "+"
    Rectangle (530,320 30x30), "0"
    Rectangle (570,320 30x30), "1"
    Rectangle (610,320 30x30), "2"
    Rectangle (490,320 30x30), "+", colour toggle: MAIN.Estacion.ProtectorBaja
        toggle MAIN.Estacion.ProtectorBaja
    Rectangle (570,320 31x31), "1", colour toggle: MAIN.Estacion.ProtectorAbajo
        toggle MAIN.Estacion.ProtectorAbajo
    Rectangle (450,360 30x30), "-"
    Rectangle (490,360 30x30), "+"
    Rectangle (530,360 30x30), "0"
    Rectangle (570,360 30x30), "1"
    Rectangle (610,360 30x30), "2"
    Rectangle (530,360 31x31), "0", colour toggle: MAIN.Estacion.PrensadorArriba
        toggle MAIN.Estacion.PrensadorArriba
    Rectangle (490,360 30x30), "+", colour toggle: MAIN.Estacion.PrensadorBaja
        toggle MAIN.Estacion.PrensadorBaja
    Rectangle (570,360 31x31), "1", colour toggle: MAIN.Estacion.PrensadorAbajoAlto
        toggle MAIN.Estacion.PrensadorAbajoAlto
    Rectangle (610,360 31x31), "2", colour toggle: MAIN.Estacion.PrensadorAbajoBajo
        toggle MAIN.Estacion.PrensadorAbajoBajo
    Rectangle (450,200 30x30), "-"
    Rectangle (450,360 30x30), "-", colour toggle: MAIN.Estacion.PrensadorSube
        toggle MAIN.Estacion.PrensadorSube
    Rectangle (490,200 30x30), "+"
    Rectangle (530,200 30x30), "0"
    Rectangle (570,200 30x30), "1"
    Rectangle (610,200 30x30), "2"
    Rectangle (490,200 30x30), "+", colour toggle: MAIN.Estacion.ManipuladorSucciona
        toggle MAIN.Estacion.ManipuladorSucciona
    Rectangle (570,200 31x31), "1", colour toggle: MAIN.Estacion.ManipuladorVacioObtenido
        toggle MAIN.Estacion.ManipuladorVacioObtenido
    Rectangle (450,400 30x30), "-"
    Rectangle (490,400 30x30), "+"
    Rectangle (530,400 30x30), "0"
    Rectangle (570,400 30x30), "1"
    Rectangle (610,400 30x30), "2"
    Rectangle (490,400 30x30), "+", colour toggle: MAIN.Estacion.HidraulicoActiva
        toggle MAIN.Estacion.HidraulicoActiva
    Rectangle (450,440 30x30), "-"
    Rectangle (490,440 30x30), "+"
    Rectangle (530,440 30x30), "0"
    Rectangle (570,440 30x30), "1"
    Rectangle (610,440 30x30), "2"
    Rectangle (490,440 30x30), "+", colour toggle: MAIN.Estacion.CintaRetenedorBaja
        toggle MAIN.Estacion.CintaRetenedorBaja
    Rectangle (450,480 30x30), "-"
    Rectangle (490,480 30x30), "+"
    Rectangle (530,480 30x30), "0"
    Rectangle (570,480 30x30), "1"
    Rectangle (610,480 30x30), "2"
    Rectangle (490,480 30x30), "+", colour toggle: MAIN.Estacion.CintaSeparadorSube
        toggle MAIN.Estacion.CintaSeparadorSube
    Rectangle (450,520 30x30), "-"
    Rectangle (450,520 30x30), "-", colour toggle: MAIN.Estacion.CintaMotorInvierte
        toggle MAIN.Estacion.CintaMotorInvierte
    Rectangle (490,520 30x30), "+"
    Rectangle (530,520 30x30), "0"
    Rectangle (570,520 30x30), "1"
    Rectangle (610,520 30x30), "2"
    Rectangle (530,520 31x31), "pp", colour toggle: MAIN.Estacion.PalePresencia
        toggle MAIN.Estacion.PalePresencia
    Rectangle (490,520 30x30), "+", colour toggle: MAIN.Estacion.CintaMotorActiva
        toggle MAIN.Estacion.CintaMotorActiva
    Rectangle (570,520 31x31), "3", colour toggle: MAIN.Estacion.CintaMotorActiva AND MAIN.Estacion.CintaMotorInvierte
    Rectangle (450,560 30x30), "-"
    Rectangle (490,560 30x30), "+"
    Rectangle (530,560 30x30), "0"
    Rectangle (570,560 30x30), "1"
    Rectangle (610,560 30x30), "2"
    Rectangle (530,560 31x31), ".2", colour toggle: MAIN.Estacion.PaleCodigoBit2
        toggle MAIN.Estacion.PaleCodigoBit2
    Rectangle (610,560 31x31), ".0", colour toggle: MAIN.Estacion.PaleCodigoBit0
        toggle MAIN.Estacion.PaleCodigoBit0
    Rectangle (570,560 31x31), ".1", colour toggle: MAIN.Estacion.PaleCodigoBit1
        toggle MAIN.Estacion.PaleCodigoBit1
    Rectangle (450,560 70x30), "%d", text variable: MAIN.Estacion.PaleCodigo
    Rectangle (610,520 31x31), "4", colour toggle: MAIN.Estacion.CintaMotorActiva AND NOT MAIN.Estacion.CintaMotorInvierte
    Rectangle (120,530 90x30), "Conectada", colour toggle: MAIN.Estacion.EstacionConectada
        toggle MAIN.Estacion.EstacionConectada
    Rectangle (120,570 90x30), "P. Marcha", colour toggle: MAIN.Estacion.PulsadorMarcha
        tap MAIN.Estacion.PulsadorMarcha
    Rectangle (120,450 90x30), "Emergencia", colour toggle: MAIN.Estacion.PulsadorEmergencia
        toggle MAIN.Estacion.PulsadorEmergencia
    Rectangle (120,650 90x30), "Manual", colour toggle: MAIN.Estacion.SelectorManual
        toggle MAIN.Estacion.SelectorManual
    Rectangle (120,610 90x30)
    Rectangle (120,610 90x30), "P. Parada", colour toggle: MAIN.Estacion.PulsadorParada
        tap MAIN.Estacion.PulsadorParada p1329445385=TRUE
    Group (56,71 119x109)
        Group (0,0 117x107)
            Polygon (119,109)
            Polygon (0,109)
            Polyline (40,94)
            Polyline (30,86)
            Polyline (30,76)
            Polyline (30,66)
            Polyline (40,54)
            Polyline (119,104)
            Polyline (119,94)
            Polyline (119,84)
            Polyline (119,74)
            Polyline (119,54)
            Rectangle (29,35 59x27)
            Rectangle (49,0 20x34)
            Rectangle (49,22 20x12)
            Rectangle (29,63 59x10)
            Polyline (40,104)
            Polyline (118,64)
            Rectangle (29,74 59x20)
        Polygon (119,109)
        Polygon (0,109)
        Polyline (40,94)
        Polyline (30,86)
        Polyline (30,76)
        Polyline (30,66)
        Polyline (40,54)
        Polyline (119,104)
        Polyline (119,94)
        Polyline (119,84)
        Polyline (119,74)
        Polyline (119,54)
        Rectangle (29,35 59x27)
        Rectangle (49,0 20x34)
        Rectangle (29,63 59x10)
        Polyline (40,104)
        Polyline (118,64)
        Rectangle (29,74 59x20)
    Rectangle (610,160 31x31), "2", colour toggle: MAIN.Estacion.ManipuladorDelante
        toggle MAIN.Estacion.ManipuladorDelante
    Group (33,615 65x21)
        tap MAIN.Estacion.AvisadorSonoro
        Rectangle (0,0 21x21)
        Polygon (5,10) (55,0) (55,0) (65,20) (5,10)
    Rectangle (660,120 210x30), "PARÁMETROS"
    Rectangle (660,150 210x290)
    Rectangle (670,160 120x30), "Hidráulico"
    Rectangle (790,160 70x30), "%s", text variable: MAIN.Estacion.TpoPrensaHidraulico
        OnMouseClick: write the text variable via Default
    Rectangle (670,200 120x30), "Protector"
    Rectangle (670,240 120x30), "Retenedor"
    Rectangle (670,280 120x30), "Separador"
    Rectangle (670,320 120x30), "Entrada Palé"
    Rectangle (670,360 120x30), "Salida Palé"
    Rectangle (670,400 120x30), "Transf. Palé"
    Rectangle (790,200 70x30), "%s", text variable: MAIN.Estacion.TpoPrensaProtector
        OnMouseClick: write the text variable via Default
    Rectangle (790,240 70x30), "%s", text variable: MAIN.Estacion.TpoCintaRetenedor
        OnMouseClick: write the text variable via Default
    Rectangle (790,280 70x30), "%s", text variable: MAIN.Estacion.TpoCintaSeparador
        OnMouseClick: write the text variable via Default
    Rectangle (790,320 70x30), "%s", text variable: MAIN.Estacion.TpoPaleEntrada
        OnMouseClick: write the text variable via Default
    Rectangle (790,360 70x30), "%s", text variable: MAIN.Estacion.TpoPaleSalida
        OnMouseClick: write the text variable via Default
    Rectangle (790,400 70x30), "%s", text variable: MAIN.Estacion.TpoPaleTransferencia
        OnMouseClick: write the text variable via Default
    Rectangle (10,200 210x30), "TAREA"
    Rectangle (10,230 210x170)
    Rectangle (120,240 90x30), "Alto", colour toggle: NOT MAIN.Estacion.RodamientoBajo
        OnMouseClick: execute { MAIN.Estacion.RodamientoBajo := FALSE; }
    Rectangle (20,280 100x30), "Solicitadas"
    Rectangle (120,280 70x30), "%d", text variable: MAIN.Estacion.UnidadesSolicitadas
        OnMouseClick: write the text variable via Default, min 1
    Rectangle (20,320 100x30), "Pendientes"
    Rectangle (120,320 70x30), "%d", text variable: MAIN.Estacion.UnidadesPendientes
        OnMouseClick: write the text variable via Default
    Rectangle (20,360 100x30), "Realizadas"
    Rectangle (120,360 70x30), "%d", text variable: MAIN.Estacion.UnidadesRealizadas
        OnMouseClick: write the text variable via Default
    Rectangle (20,240 90x30), "Bajo", colour toggle: MAIN.Estacion.RodamientoBajo
        OnMouseClick: execute { MAIN.Estacion.RodamientoBajo := TRUE; }
    Rectangle (660,450 210x240)
    Rectangle (450,160 30x30), "-", colour toggle: MAIN.Estacion.ManipuladorAtras
        toggle MAIN.Estacion.ManipuladorAtras
    RoundedRectangle (670,705 60x20), "CI"
    RoundedRectangle (670,705 60x20), "CI", colour toggle: MAIN.Estacion.CondicionInicial, invisible if: NOT MAIN.Estacion.Coordinador.Ready
    RoundedRectangle (740,705 60x20), "Reset", colour toggle: MAIN.Estacion.EstadoReinicia, invisible if: NOT MAIN.FMS203.Reposo
        tap MAIN.Estacion.EstadoReinicia
    RoundedRectangle (600,705 60x20), "Reposo", colour toggle: MAIN.Estacion.Coordinador.Ready
    Rectangle (190,280 20x31), "1"
        OnMouseClick: execute { MAIN.Estacion.UnidadesSolicitadas := 1 }
    Rectangle (190,320 20x30), "0"
        OnMouseClick: execute { MAIN.Estacion.UnidadesPendientes := 0 }
    Rectangle (190,360 20x30), "0"
        OnMouseClick: execute { MAIN.Estacion.UnidadesRealizadas := 0 }
    RoundedRectangle (810,705 60x20), "Pausa", colour toggle: MAIN.Estacion.EstadoPausa, invisible if: NOT MAIN.FMS203.Reposo
        toggle MAIN.Estacion.EstadoPausa
    Rectangle (230,60 640x50)
    Rectangle (240,70 120x30), "Modo"
    Rectangle (370,70 70x30), "%s", text variable: MAIN.Estacion.Director.Modo
    Rectangle (450,70 410x30), "%s", text list: 'ModoDescripcion', text index: MAIN.Estacion.Director.Modo
    Rectangle (20,15 120x30), "FMS-203"
END_VISUALIZATION
